(* IEC 61131-3 sources: generating_plc_code_with_llms/Code#1/ChatGPT_3.5/second run, 20 files *)

(* ---- 10.st ---- *)
//6.25
//4
FUNCTION Sigmoid: REAL
VAR_INPUT
    x: REAL;  // Input value
END_VAR

VAR
    e_to_power_minus_x: REAL;
END_VAR

BEGIN
    e_to_power_minus_x := EXP(-x);
    Sigmoid := 1 / (1 + e_to_power_minus_x);
END_FUNCTION

(* ---- 11.st ---- *)
//7.44s
//4
FUNCTION Sign: INT
VAR_INPUT
    x: REAL;  // Input value
END_VAR

VAR
    sign_result: INT := 0;
END_VAR

BEGIN
    IF x > 0.0 THEN
        sign_result := 1;
    ELSIF x < 0.0 THEN
        sign_result := -1;
    ELSE
        sign_result := 0;
    END_IF

    Sign := sign_result;
END_FUNCTION

(* ---- 12.st ---- *)
//7.32s
//4
FUNCTION HyperbolicSine: REAL
VAR_INPUT
    x: REAL;  // Input value
END_VAR

VAR
    sinh_result: REAL;
END_VAR

BEGIN
    sinh_result := (EXP(x) - EXP(-x)) / 2.0;
    HyperbolicSine := sinh_result;
END_FUNCTION

(* ---- 14.st ---- *)
// 27.5s
// 3
FUNCTION FC1001
VAR_INPUT
    MeasuredValue: REAL;           // Measured value from the sensor
    SwitchingValue: REAL;          // Predeterminable switching value
    HysteresisPercentage: REAL;    // Switching hysteresis in % of the switching value
    SwitchedOn: BOOL;              // Output indicating if the output should be switched on or off
END_VAR

VAR
    SwitchingThresholdHigh: REAL;  // Threshold for switching on
    SwitchingThresholdLow: REAL;   // Threshold for switching off
    OutputState: BOOL;             // Current state of the output
END_VAR

BEGIN
    // Calculate switching thresholds based on the hysteresis
    SwitchingThresholdHigh := SwitchingValue * (1 + HysteresisPercentage / 100.0);
    SwitchingThresholdLow := SwitchingValue * (1 - HysteresisPercentage / 100.0);

    // Determine the output state based on the measured value and thresholds
    IF MeasuredValue > SwitchingThresholdHigh THEN
        OutputState := TRUE;  // Switched on
    ELSIF MeasuredValue < SwitchingThresholdLow THEN
        OutputState := FALSE; // Switched off
    END_IF

    // Update the output state based on the control input
    IF SwitchedOn THEN
        OutputState := TRUE;
    ELSE
        OutputState := FALSE;
    END_IF

    // Return the current state of the output
    FC1001 := OutputState;
END_FUNCTION

(* ---- 15.st ---- *)
// 26.41s
// 4
FUNCTION FC1002
VAR_INPUT
    E_A: BOOL;       // Switch for turning on/off the monitoring system
    UltrasonicDetected: BOOL;  // Ultrasonic sensor detection signal
    P1: BOOL;        // Status indicating the monitoring system is switched on
END_VAR

VAR
    Timer: TON;      // Timer to measure the duration of detection
    P_HU: BOOL;      // Acoustic warning signal
    P_AL: BOOL;      // Alarm signal
    TimerDuration: TIME := T#3S;  // Duration for the alarm timer
END_VAR

BEGIN
    // Initialize the timer parameters
    Timer(IN := UltrasonicDetected AND E_A, PT := TimerDuration);

    // Output signals initialization
    P_HU := FALSE;
    P_AL := FALSE;

    // Check if the monitoring system is switched on
    IF E_A THEN
        P1 := TRUE;  // Monitoring system is switched on

        // Check if the ultrasonic sensor detects an approach
        IF UltrasonicDetected THEN
            // Start the timer when an approach is detected
            Timer(IN := TRUE);

            // If the timer reaches the specified duration, switch off the warning signal
            IF Timer.Q THEN
                P_HU := FALSE;

                // Switch on the alarm signal
                P_AL := TRUE;
            ELSE
                // If the detection is within the timer duration, switch on the warning signal
                P_HU := TRUE;

                // Switch off the alarm signal
                P_AL := FALSE;
            END_IF
        END_IF
    ELSE
        // Switch off all signals when the monitoring system is switched off
        P1 := FALSE;
        P_HU := FALSE;
        P_AL := FALSE;
    END_IF
END_FUNCTION

(* ---- 18.st ---- *)
// 32.44s
// 4
FUNCTION FC1003
VAR_INPUT
    DigitalInput: INT;  // Digital input value from the temperature sensor (0 to 255)
    IN_MIN: INT;        // Lower limit of the digital input range
    IN_MAX: INT;        // Upper limit of the digital input range
    OUT_MIN: REAL;      // Lower limit of the output temperature range
    OUT_MAX: REAL;      // Upper limit of the output temperature range
END_VAR

VAR_OUTPUT
    Temperature: REAL;  // Converted temperature value
END_VAR

VAR
    M: REAL;            // Slope of the linear interpolation
    C: REAL;            // Y-intercept of the linear interpolation
END_VAR

BEGIN
    // Ensure that the input limits are not equal to avoid division by zero
    IF IN_MIN <> IN_MAX THEN
        // Calculate the slope and y-intercept for linear interpolation
        M := (OUT_MAX - OUT_MIN) / (IN_MAX - IN_MIN);
        C := OUT_MIN - M * IN_MIN;

        // Perform linear interpolation to map the digital input to temperature
        Temperature := M * DigitalInput + C;
    ELSE
        // If input limits are equal, set Temperature to OUT_MIN
        Temperature := OUT_MIN;
    END_IF
END_FUNCTION

(* ---- 2.st ---- *)
// 8.03s
//2
FUNCTION CalculateBinomialCoefficient: INT
VAR_INPUT
    n: INT;  // The total number of items (n)
    k: INT;  // The number of items to choose (k)
END_VAR

VAR
    result: INT;
    i: INT;
    nFactorial: INT := 1;  // Initialize n! to 1
    kFactorial: INT := 1;  // Initialize k! to 1
END_VAR

BEGIN
    result := 0;

    IF n >= k THEN
        FOR i := 1 TO n DO
            nFactorial := nFactorial * i;
        END_FOR

        FOR i := 1 TO k DO
            kFactorial := kFactorial * i;
        END_FOR

        result := nFactorial / (kFactorial * (n - k)!);
    END_IF

    RETURN result;
END_FUNCTION

(* ---- 3.st ---- *)
//5.75s
//2
FUNCTION CalculateFibonacci: INT
VAR_INPUT
    n: INT;  // The position of the Fibonacci number to calculate
END_VAR

VAR
    result: INT;
END_VAR

BEGIN
    IF n <= 0 THEN
        result := 0;
    ELSIF n = 1 THEN
        result := 1;
    ELSE
        result := CalculateFibonacci(n - 1) + CalculateFibonacci(n - 2);
    END_IF

    RETURN result;
END_FUNCTION

(* ---- 19.st ---- *)
// 17.9s
// 3
FUNCTION_BLOCK FB1005
VAR_INPUT
    START: BOOL;       // Start of the measurement (connected to sensor S1)
    THICKNESS: REAL;   // Input representing the difference between two laser measurements
    V_MAX: REAL;       // Maximum allowed thickness
    V_MIN: REAL;       // Minimum allowed thickness
END_VAR

VAR_OUTPUT
    D_MAX: REAL;       // Largest plate thickness value
    D_MIN: REAL;       // Smallest plate thickness value
    P1: BOOL;          // Reject light signal
END_VAR

VAR
    SensorActive: BOOL := FALSE;  // Flag indicating if the sensor is active
    TempD_MAX: REAL := 0.0;       // Temporary storage for the largest value
    TempD_MIN: REAL := 0.0;       // Temporary storage for the smallest value
END_VAR

METHOD CheckThickness : BOOL
    IF SensorActive THEN
        // During and after the measurement
        D_MAX := TempD_MAX;
        D_MIN := TempD_MIN;

        // Check if values are outside the tolerance band
        IF (D_MAX > V_MAX OR D_MIN < V_MIN) THEN
            P1 := TRUE;  // Switch on reject light
        ELSE
            P1 := FALSE; // Switch off reject light
        END_IF

        // Reset temporary storage at the end of the measurement
        IF NOT START THEN
            TempD_MAX := THICKNESS;
            TempD_MIN := THICKNESS;
            SensorActive := FALSE;
        END_IF

        // Output the result of the thickness check
        CheckThickness := TRUE;
    ELSE
        // At the start of a new measurement
        SensorActive := START;

        // Initialize temporary storage at the start of a new measurement
        IF SensorActive THEN
            TempD_MAX := THICKNESS;
            TempD_MIN := THICKNESS;
        END_IF

        // Output the result of the thickness check
        CheckThickness := FALSE;
    END_IF
END_METHOD
END_FUNCTION_BLOCK

(* ---- 21.st ---- *)
// 64.68s
// weiter generieren
// 2
FUNCTION_BLOCK BURNER
VAR_INPUT
    IN: BOOL;                 // Control input to start the burner
    OVER_TEMP: BOOL;          // Boiler thermostat protection
    OIL_TEMP: BOOL;           // Signal indicating the oil temperature is reached
    MULTIPLE_IGNITION: BOOL;  // Enable multiple ignitions after flame failure
    STAGE2: BOOL;             // Input to activate the second stage
    RST: BOOL;                // Reset input to restart the operation after lockout time
END_VAR

VAR_OUTPUT
    PRE_HEAT: BOOL;         // Output to start fuel oil warming
    MOTOR_ON: BOOL;         // Output to activate the motor
    FAN_ON: BOOL;           // Output to activate the fan
    IGNITION_ON: BOOL;      // Output to activate the ignition
    OIL_VALVE_OPEN: BOOL;   // Output to open the oil valve
    STATUS: INT;            // Output status indicating the current state of the module
    FAIL: BOOL;             // Output indicating a failure
END_VAR

VAR
    PRE_HEAT_TIMER: TON;                // Timer for fuel oil warming
    PRE_VENT_TIMER: TON;                // Timer for pre-purge (pre-ventilation)
    IGNITION_TIMER: TON;                // Timer for ignition
    SAFETY_TIMER: TON;                  // Timer for safety time
    POST_IGNITION_TIMER: TON;           // Timer for post-ignition time
    STAGE2_DELAY_TIMER: TON;            // Timer for delay before activating stage 2
    LOCKOUT_TIMER: TON;                 // Timer for lockout time after a fault
    OPERATION_TIMER: TON := T#0S;       // Timer for measuring the overall operation time
    STAGE1_OPERATION_TIMER: TON := T#0S; // Timer for measuring stage 1 operation time
    STAGE2_OPERATION_TIMER: TON := T#0S; // Timer for measuring stage 2 operation time

    PRE_HEAT_TIME: TIME := T#5S;         // Pre-heating time
    PRE_VENTILATION_TIME: TIME := T#10S; // Pre-ventilation time
    PPR_IGNITION_TIME: TIME := T#5S;     // Time before opening the oil valve during ignition
    SAFETY_TIME: TIME := T#10S;           // Safety time
    POST_IGNITION_TIME: TIME := T#5S;    // Post-ignition time
    STAGE2_DELAY: TIME := T#60S;         // Delay before activating stage 2
    LOCKOUT_TIME: TIME := T#300S;        // Lockout time after a fault

    STANDBY: INT := 110;     // Standby state
    STARTUP: INT := 111;     // Startup state
    STAGE1_RUNNING: INT := 112;  // Burner running on stage 1 state
    STAGE2_RUNNING: INT := 113;  // Burner running on stage 2 state
    ERROR_FUEL_WARMING: INT := 1;  // Error: Fuel oil warming not responded within PRE_HEAT_TIME
    ERROR_FAME_SENSOR_PRE_HEAT: INT := 2;  // Error: Fame sensor active during fuel oil warming
    ERROR_FAME_SENSOR_VENT: INT := 3;  // Error: Fame sensor active during pre-ventilation
    ERROR_SAFETY_TIME: INT := 4;  // Error: Safety time passed without fame
    ERROR_FAME_STOPS: INT := 5;  // Error: Fame stops in operation
    ERROR_OVERHEATING: INT := 9;  // Error: Boiler overheating contact has tripped
END_VAR

METHOD BurnerControl : BOOL
    CASE STATUS OF
        STANDBY:
            IF IN AND NOT OVER_TEMP THEN
                // Start the fuel oil warming
                PRE_HEAT := TRUE;
                STATUS := STARTUP;
                OPERATION_TIMER(IN := TRUE);
            ELSE
                // Standby state
                STATUS := STANDBY;
            END_IF;
        STARTUP:
            // Fuel oil warming
            IF PRE_HEAT_TIMER.Q THEN
                // Check if fuel oil warming has responded within PRE_HEAT_TIME
                FAIL := TRUE;
                STATUS := ERROR_FUEL_WARMING;
            ELSIF OIL_TEMP AND NOT PRE_VENT_TIMER.Q THEN
                // Start the motor and fan after fuel oil warming
                MOTOR_ON := TRUE;
                FAN_ON := TRUE;
                STATUS := STAGE1_RUNNING;
                STAGE1_OPERATION_TIMER(IN := TRUE);
            END_IF;
        STAGE1_RUNNING:
            // Check if fame sensor is active during fuel oil warming
            IF IGNITION_ON AND PRE_HEAT_TIMER.Q THEN
                FAIL := TRUE;
                STATUS := ERROR_FAME_SENSOR_PRE_HEAT;
            ELSIF IGNITION_ON AND PRE_VENT_TIMER.Q THEN
                // Check if fame sensor is active during pre-ventilation
                FAIL := TRUE;
                STATUS := ERROR_FAME_SENSOR_VENT;
            ELSIF SAFETY_TIMER.Q THEN
                // Check if safety time has passed without fame
                FAIL := TRUE;
                STATUS := ERROR_SAFETY_TIME;
            ELSIF NOT IGNITION_ON AND POST_IGNITION_TIMER.Q THEN
                // Check if fame stops in operation
                FAIL := TRUE;
                STATUS := ERROR_FAME_STOPS;
            ELSIF OVER_TEMP THEN
                // Check if boiler overheating protection is active
                STATUS := ERROR_OVERHEATING;
            ELSIF STAGE2 AND STAGE2_DELAY_TIMER.Q THEN
                // Activate stage 2 after the delay
                STATUS := STAGE2_RUNNING;
                STAGE2_OPERATION_TIMER(IN := TRUE);
            END_IF;
        STAGE2_RUNNING:
            // Continue with stage 2 operation
            // (Additional logic for stage 2 can be added here)
            // ...
            IF OVER_TEMP THEN
                // Check if boiler overheating protection is active
                STATUS := ERROR_OVERHEATING;
            END_IF;
    END_CASE;

    // Check if the burner is in lockout state
    IF LOCKOUT_TIMER.Q THEN
        STATUS := 0;  // Reset the status to indicate the lockout state
        FAIL := FALSE;  // Reset the fail flag
    END_IF;

    // Reset the operation timer if the burner is not in operation
    IF STATUS = STANDBY OR STATUS = 0 THEN
        OPERATION_TIMER(IN := FALSE);
    END_IF;

    // Check for reset condition to restart the operation after lockout time
    IF NOT RST AND LOCKOUT_TIMER.Q THEN
        LOCKOUT_TIMER(IN := FALSE);
    ELSIF RST THEN
        LOCKOUT_TIMER(IN := TRUE, PT := LOCKOUT_TIME);
    END_IF;

    // Output status indicating the current state of the module
    BurnerControl := TRUE;
END_METHOD
END_FUNCTION_BLOCK

(* ---- 1.st ---- *)
//5.24s
//2
PROGRAM AlarmControl
VAR
    xAlarm1: BOOL := FALSE;
    xAlarm2: BOOL := FALSE;
    xAllOn: BOOL := FALSE;
    xAllOff: BOOL := FALSE;
END_VAR

METHOD SetAlarms: BOOL
    IF xAllOn THEN
        xAlarm1 := TRUE;
        xAlarm2 := TRUE;
    ELSIF xAllOff THEN
        xAlarm1 := FALSE;
        xAlarm2 := FALSE;
    END_IF
    RETURN TRUE;
END_METHOD

METHOD TurnOffAlarms
    xAlarm1 := FALSE;
    xAlarm2 := FALSE;
END_METHOD

END_PROGRAM

(* ---- 13.st ---- *)
//8.97s
//2
PROGRAM NumberSearch
VAR
    Numbers: ARRAY[1..100] OF INT;  // List of 100 random numbers
    NumberToFind: INT := 10;  // The number to find
    Found: BOOL := FALSE;  // Flag to indicate if the number is found
END_VAR

BEGIN
    // Initialize the list of 100 random numbers (simulated)
    FOR i := 1 TO 100 DO
        Numbers[i] := RANDOM(0, 100);  // Replace with actual random number generation
    END_FOR

    // Search for the number 10 in the list
    REPEAT
        FOR i := 1 TO 100 DO
            IF Numbers[i] = NumberToFind THEN
                Found := TRUE;
                EXIT;  // Abort the search if the number is found
            END_IF
        END_FOR
        EXIT;  // Abort the search if the end of the list is reached
    UNTIL FALSE;

    // Check if the number was found or not
    IF Found THEN
        // Number 10 was found in the list
        // Implement the necessary actions when the number is found
    ELSE
        // Number 10 was not found in the list
        // Implement the necessary actions when the number is not found
    END_IF
END_PROGRAM

(* ---- 16.st ---- *)
//10.81s
//2
PROGRAM TrafficLightControl
VAR
    North_green: BOOL := TRUE;  // North green light
    North_yellow: BOOL := FALSE;  // North yellow light
    North_red: BOOL := FALSE;  // North red light
    East_green: BOOL := FALSE;  // East green light
    East_yellow: BOOL := FALSE;  // East yellow light
    East_red: BOOL := TRUE;  // East red light
    Timer: TON;  // Timer to control the light cycle
END_VAR

BEGIN
    // Initialize the timer parameters
    Timer(IN := TRUE, PT := T#5000ms);

    // Control the traffic light cycle
    IF Timer.Q THEN
        // First 5000ms - North green, East red
        North_green := TRUE;
        North_yellow := FALSE;
        North_red := FALSE;
        East_green := FALSE;
        East_yellow := FALSE;
        East_red := TRUE;
    ELSIF Timer.ET THEN
        // 5000ms to 5500ms - North yellow, East red
        North_green := FALSE;
        North_yellow := TRUE;
        North_red := FALSE;
        East_green := FALSE;
        East_yellow := FALSE;
        East_red := TRUE;
    ELSIF Timer.Q2 THEN
        // 5500ms to 9500ms - North red, East green
        North_green := FALSE;
        North_yellow := FALSE;
        North_red := TRUE;
        East_green := TRUE;
        East_yellow := FALSE;
        East_red := FALSE;
    ELSIF Timer.ET2 THEN
        // 9500ms to 10000ms - North red, East yellow
        North_green := FALSE;
        North_yellow := FALSE;
        North_red := TRUE;
        East_green := FALSE;
        East_yellow := TRUE;
        East_red := FALSE;
    END_IF
END_PROGRAM

(* ---- 17.st ---- *)
//16.93s
//2
PROGRAM WeatherStation
VAR
    TemperatureSensorValue: INT := 0;  // Analog input value for temperature (0 - 32767)
    HumiditySensorValue: INT := 0;  // Analog input value for humidity (0 - 32767)
    TemperatureText: STRING := "";  // Text to display temperature condition
END_VAR

BEGIN
    // Simulate reading temperature and humidity values from analog inputs
    // Replace with actual analog input readings in your system
    TemperatureSensorValue := 22000;  // Example temperature reading
    HumiditySensorValue := 5000;     // Example humidity reading

    // Evaluate temperature condition
    IF TemperatureSensorValue < 18000 THEN
        TemperatureText := "Cold";
    ELSIF TemperatureSensorValue >= 18000 AND TemperatureSensorValue <= 25000 THEN
        // Temperature is in the optimum range (18 - 25°C), evaluate humidity
        IF HumiditySensorValue >= 4000 AND HumiditySensorValue <= 7500 THEN
            TemperatureText := "Opt";
        ELSE
            TemperatureText := "Temp. OK";
        END_IF
    ELSE
        TemperatureText := "Hot";
    END_IF

    // Display the temperature condition text inside the house
    // The value of TemperatureText can be displayed as needed
END_PROGRAM

(* ---- 20.st ---- *)
// 16.52s
// 4
PROGRAM InterlockProgram
VAR
    I1: BOOL;      // Input for Q1
    I2: BOOL;      // Input for Q2
    Q1: BOOL;      // Output Q1
    Q2: BOOL;      // Output Q2
    TL: TIME := T#1S;  // Dead time between the two outputs
    TimerQ1: TON;   // Timer for Q1
    TimerQ2: TON;   // Timer for Q2
END_VAR

VAR CONSTANT
    TRUE_TIME: TIME := T#0S;  // Constant representing TRUE for a timer
END_VAR

BEGIN
    // Interlock logic for Q1
    IF NOT Q2 AND I1 THEN
        // Start the timer for Q1 if Q2 is FALSE and I1 is TRUE
        TimerQ1(IN := TRUE, PT := TL);
        // Set Q1 to TRUE if the timer for Q1 has elapsed
        Q1 := TimerQ1.Q;
    ELSE
        // Reset the timer for Q1 if Q2 is TRUE or I1 is FALSE
        TimerQ1(IN := FALSE);
        // Set Q1 to FALSE
        Q1 := FALSE;
    END_IF

    // Interlock logic for Q2
    IF NOT Q1 AND I2 THEN
        // Start the timer for Q2 if Q1 is FALSE and I2 is TRUE
        TimerQ2(IN := TRUE, PT := TL);
        // Set Q2 to TRUE if the timer for Q2 has elapsed
        Q2 := TimerQ2.Q;
    ELSE
        // Reset the timer for Q2 if Q1 is TRUE or I2 is FALSE
        TimerQ2(IN := FALSE);
        // Set Q2 to FALSE
        Q2 := FALSE;
    END_IF
END_PROGRAM

(* ---- 4.st ---- *)
//14.32s
//2
PROGRAM FillLevelMonitor
VAR
    FillLevelAnalog: INT;  // Analog value (0 - 32767)
    FillLevelPercent: REAL;  // Fill level in percentage (0-100%)
    LowLevel: BOOL := FALSE;  // Output for low fill level
    OkLevel: BOOL := FALSE;   // Output for ok fill level
    HighLevel: BOOL := FALSE; // Output for high fill level
    WarningHorn: BOOL := FALSE; // Output for warning horn
END_VAR

BEGIN
    // Read the analog fill level value (0 - 32767), e.g., from a sensor
    FillLevelAnalog := YourAnalogInputValue;

    // Convert the analog fill level to a percentage (0-100%)
    FillLevelPercent := (REAL(FillLevelAnalog) / 32767.0) * 100.0;

    // Use the CASE instruction to categorize the fill level
    CASE
        FillLevelPercent < 1.0:
            LowLevel := TRUE;
            OkLevel := FALSE;
            HighLevel := FALSE;
            WarningHorn := TRUE;
        FillLevelPercent >= 1.0 AND FillLevelPercent <= 70.0:
            LowLevel := FALSE;
            OkLevel := TRUE;
            HighLevel := FALSE;
            WarningHorn := FALSE;
        FillLevelPercent > 70.0:
            LowLevel := FALSE;
            OkLevel := FALSE;
            HighLevel := TRUE;
            WarningHorn := FALSE;
    END_CASE;
END_PROGRAM

(* ---- 5.st ---- *)
//10.68s
//2
PROGRAM GateController
VAR
    Start_Loop: BOOL := TRUE;  // Start the loop (initially TRUE)
    One_Hour_Timer: TIME := T#1H;  // One-hour timer
    Gate_Open: BOOL := FALSE;  // Gate status (initially closed)
    Auth_String: STRING := "my_defined_str";  // Expected authentication string
    App_Presence: BOOL := FALSE;  // App presence indicator
    Car_Presence: BOOL := FALSE;  // Car presence indicator
END_VAR

BEGIN
    // If the timer is not running and Start_Loop is FALSE, start the timer
    IF NOT One_Hour_Timer.RUNNING AND NOT Start_Loop THEN
        One_Hour_Timer(IN := TRUE);
    END_IF

    // Check if the timer has timed out and the gate is open
    IF One_Hour_Timer.Q AND Gate_Open THEN
        Gate_Open := FALSE;  // Close the gate
    END_IF

    // Check for authentication conditions (app presence and matching Auth_String)
    IF App_Presence AND Auth_String = "my_defined_str" THEN
        Gate_Open := TRUE;  // Open the gate
    END_IF
END_PROGRAM

(* ---- 6.st ---- *)
//13.18
//3
PROGRAM CraneLift
VAR
    doConvTop: BOOL := FALSE;  // Conveyor belt control for top conveyor
    doConvBottom: BOOL := FALSE;  // Conveyor belt control for bottom conveyor
    diConvTop: BOOL := FALSE;  // Light barrier for top conveyor
    diConvBottom: BOOL := FALSE;  // Light barrier for bottom conveyor
    doLiftTop: BOOL := FALSE;  // Lift control for the top position
    doLiftBottom: BOOL := FALSE;  // Lift control for the bottom position
    diLiftTop: BOOL := FALSE;  // Lift position sensor for the top position
    diLiftBottom: BOOL := FALSE;  // Lift position sensor for the bottom position
    doConvLift: BOOL := FALSE;  // Lift conveyor belt control
    diBoxLift: BOOL := FALSE;  // Crate sensor on the lift conveyor
    doLiftUnload: BOOL := FALSE;  // Lift control for unloading position
    diLiftUnload: BOOL := FALSE;  // Lift position sensor for unloading position
END_VAR

BEGIN
    // If the light barrier for the top conveyor is activated, stop the top conveyor
    IF diConvTop THEN
        doConvTop := FALSE;
    END_IF

    // If the light barrier for the bottom conveyor is activated, stop the bottom conveyor
    IF diConvBottom THEN
        doConvBottom := FALSE;
    END_IF

    // Request the lift to the top position if not already requested
    IF diConvTop AND NOT diLiftTop THEN
        doLiftTop := TRUE;
    END_IF

    // Request the lift to the bottom position if not already requested
    IF diConvBottom AND NOT diLiftBottom THEN
        doLiftBottom := TRUE;
    END_IF

    // If the lift has reached the requested top position, start the lift conveyor belt
    IF diLiftTop AND NOT diBoxLift THEN
        doConvLift := TRUE;
    END_IF

    // If the crate is detected on the lift conveyor, stop the lift conveyor belt
    IF diBoxLift THEN
        doConvLift := FALSE;
    END_IF

    // Request the lift to the unloading position if not already requested
    IF diBoxLift AND NOT diLiftUnload THEN
        doLiftUnload := TRUE;
    END_IF

    // If the lift has reached the unloading position, start unloading the crate onto the unloading conveyor
    IF diLiftUnload THEN
        doLiftUnload := FALSE;
        // Perform actions to unload the crate onto the unloading conveyor
    END_IF
END_PROGRAM

(* ---- 7.st ---- *)
//10.15s
//2
PROGRAM CraneLoadCalculation
VAR
    LoadReceptorValues: ARRAY[1..5] OF INT;  // Load receptor values (0 - 32767)
    TotalLoad: REAL := 0.0;  // Total load variable
    AverageLoad: REAL := 0.0;  // Average load variable
    NumLoadReceptors: INT := 5;  // Number of load receptors (constant)
END_VAR

VAR CONSTANT
    LoadValueMax: INT := 32767;  // Maximum load value (constant)
END_VAR

VAR CONSTANT
    TotalLoadDivider: INT := 1000;  // Constant used for calculating average load
END_VAR

BEGIN
    // Simulate reading values from the load receptors
    // In practice, you would read the actual analog input values here
    LoadReceptorValues[1] := 15000;
    LoadReceptorValues[2] := 20000;
    LoadReceptorValues[3] := 25000;
    LoadReceptorValues[4] := 28000;
    LoadReceptorValues[5] := 32000;

    // Calculate the total load using a FOR loop
    FOR i := 1 TO NumLoadReceptors DO
        TotalLoad := TotalLoad + REAL(LoadReceptorValues[i]);
    END_FOR

    // Calculate the average load
    IF NumLoadReceptors > 0 THEN
        AverageLoad := TotalLoad / (NumLoadReceptors * TotalLoadDivider);
    ELSE
        AverageLoad := 0.0;
    END_IF
END_PROGRAM

(* ---- 9.st ---- *)
//7.03s
//4
PROGRAM LeapYearCheck
VAR
    YEAR: INT;  // Input year to be checked
    IsLeapYear: BOOL := FALSE;  // Output indicating if it's a leap year
END_VAR

BEGIN
    // Check if the given year is a leap year
    IF (YEAR MOD 4 = 0) AND ((YEAR MOD 100 <> 0) OR (YEAR MOD 400 = 0)) THEN
        IsLeapYear := TRUE;
    ELSE
        IsLeapYear := FALSE;
    END_IF
END_PROGRAM
